Error[1788].CreateEx(TC_Events.Error.Error1788,FALSE,0);
Error[1789].CreateEx(TC_Events.Error.Error1789,FALSE,0);
Error[1790].CreateEx(TC_Events.Error.Error1790,FALSE,0);
Error[1791].CreateEx(TC_Events.Error.Error1791,FALSE,0);
Error[1792].CreateEx(TC_Events.Error.Error1792,FALSE,0);
Error[1793].CreateEx(TC_Events.Error.Error1793,FALSE,0);
Error[1794].CreateEx(TC_Events.Error.Error1794,FALSE,0);
Error[1795].CreateEx(TC_Events.Error.Error1795,FALSE,0);
Error[1796].CreateEx(TC_Events.Error.Error1796,FALSE,0);
Error[1797].CreateEx(TC_Events.Error.Error1797,FALSE,0);
Error[1798].CreateEx(TC_Events.Error.Error1798,FALSE,0);
Error[1799].CreateEx(TC_Events.Error.Error1799,FALSE,0);
Error[1800].CreateEx(TC_Events.Error.Error1800,FALSE,0);
Error[1801].CreateEx(TC_Events.Error.Error1801,FALSE,0);
Error[1802].CreateEx(TC_Events.Error.Error1802,FALSE,0);
Error[1803].CreateEx(TC_Events.Error.Error1803,FALSE,0);
Error[1804].CreateEx(TC_Events.Error.Error1804,FALSE,0);
Error[1805].CreateEx(TC_Events.Error.Error1805,FALSE,0);
Error[1806].CreateEx(TC_Events.Error.Error1806,FALSE,0);
Error[1807].CreateEx(TC_Events.Error.Error1807,FALSE,0);
Error[1808].CreateEx(TC_Events.Error.Error1808,FALSE,0);
Error[1809].CreateEx(TC_Events.Error.Error1809,FALSE,0);
Error[1810].CreateEx(TC_Events.Error.Error1810,FALSE,0);
Error[1811].CreateEx(TC_Events.Error.Error1811,FALSE,0);
Error[1812].CreateEx(TC_Events.Error.Error1812,FALSE,0);
Error[1813].CreateEx(TC_Events.Error.Error1813,FALSE,0);
Error[1814].CreateEx(TC_Events.Error.Error1814,FALSE,0);
Error[1815].CreateEx(TC_Events.Error.Error1815,FALSE,0);
Error[1816].CreateEx(TC_Events.Error.Error1816,FALSE,0);
Error[1817].CreateEx(TC_Events.Error.Error1817,FALSE,0);
Error[1818].CreateEx(TC_Events.Error.Error1818,FALSE,0);
Error[1819].CreateEx(TC_Events.Error.Error1819,FALSE,0);
Error[1820].CreateEx(TC_Events.Error.Error1820,FALSE,0);
Error[1821].CreateEx(TC_Events.Error.Error1821,FALSE,0);
Error[1822].CreateEx(TC_Events.Error.Error1822,FALSE,0);
Error[1823].CreateEx(TC_Events.Error.Error1823,FALSE,0);
Error[1824].CreateEx(TC_Events.Error.Error1824,FALSE,0);
Error[1825].CreateEx(TC_Events.Error.Error1825,FALSE,0);
Error[1826].CreateEx(TC_Events.Error.Error1826,FALSE,0);
Error[1827].CreateEx(TC_Events.Error.Error1827,FALSE,0);
Error[1828].CreateEx(TC_Events.Error.Error1828,FALSE,0);
Error[1829].CreateEx(TC_Events.Error.Error1829,FALSE,0);
Error[1830].CreateEx(TC_Events.Error.Error1830,FALSE,0);
Error[1831].CreateEx(TC_Events.Error.Error1831,FALSE,0);
Error[1832].CreateEx(TC_Events.Error.Error1832,FALSE,0);
Error[1833].CreateEx(TC_Events.Error.Error1833,FALSE,0);
Error[1834].CreateEx(TC_Events.Error.Error1834,FALSE,0);
Error[1835].CreateEx(TC_Events.Error.Error1835,FALSE,0);
Error[1836].CreateEx(TC_Events.Error.Error1836,FALSE,0);
Error[1837].CreateEx(TC_Events.Error.Error1837,FALSE,0);
Error[1838].CreateEx(TC_Events.Error.Error1838,FALSE,0);
Error[1839].CreateEx(TC_Events.Error.Error1839,FALSE,0);
Error[1840].CreateEx(TC_Events.Error.Error1840,FALSE,0);
Error[1841].CreateEx(TC_Events.Error.Error1841,FALSE,0);
Error[1842].CreateEx(TC_Events.Error.Error1842,FALSE,0);
Error[1843].CreateEx(TC_Events.Error.Error1843,FALSE,0);
Error[1844].CreateEx(TC_Events.Error.Error1844,FALSE,0);
Error[1845].CreateEx(TC_Events.Error.Error1845,FALSE,0);
Error[1846].CreateEx(TC_Events.Error.Error1846,FALSE,0);
Error[1847].CreateEx(TC_Events.Error.Error1847,FALSE,0);
Error[1848].CreateEx(TC_Events.Error.Error1848,FALSE,0);
Error[1849].CreateEx(TC_Events.Error.Error1849,FALSE,0);
Error[1850].CreateEx(TC_Events.Error.Error1850,FALSE,0);
Error[1851].CreateEx(TC_Events.Error.Error1851,FALSE,0);
Error[1852].CreateEx(TC_Events.Error.Error1852,FALSE,0);
Error[1853].CreateEx(TC_Events.Error.Error1853,FALSE,0);
Error[1854].CreateEx(TC_Events.Error.Error1854,FALSE,0);
Error[1855].CreateEx(TC_Events.Error.Error1855,FALSE,0);
Error[1856].CreateEx(TC_Events.Error.Error1856,FALSE,0);
Error[1857].CreateEx(TC_Events.Error.Error1857,FALSE,0);
Error[1858].CreateEx(TC_Events.Error.Error1858,FALSE,0);
Error[1859].CreateEx(TC_Events.Error.Error1859,FALSE,0);
Error[1860].CreateEx(TC_Events.Error.Error1860,FALSE,0);
Error[1861].CreateEx(TC_Events.Error.Error1861,FALSE,0);
Error[1862].CreateEx(TC_Events.Error.Error1862,FALSE,0);
Error[1863].CreateEx(TC_Events.Error.Error1863,FALSE,0);
Error[1864].CreateEx(TC_Events.Error.Error1864,FALSE,0);
Error[1865].CreateEx(TC_Events.Error.Error1865,FALSE,0);
Error[1866].CreateEx(TC_Events.Error.Error1866,FALSE,0);
Error[1867].CreateEx(TC_Events.Error.Error1867,FALSE,0);
Error[1868].CreateEx(TC_Events.Error.Error1868,FALSE,0);
Error[1869].CreateEx(TC_Events.Error.Error1869,FALSE,0);
Error[1870].CreateEx(TC_Events.Error.Error1870,FALSE,0);
Error[1871].CreateEx(TC_Events.Error.Error1871,FALSE,0);
Error[1872].CreateEx(TC_Events.Error.Error1872,FALSE,0);
Error[1873].CreateEx(TC_Events.Error.Error1873,FALSE,0);
Error[1874].CreateEx(TC_Events.Error.Error1874,FALSE,0);
Error[1875].CreateEx(TC_Events.Error.Error1875,FALSE,0);
Error[1876].CreateEx(TC_Events.Error.Error1876,FALSE,0);
Error[1877].CreateEx(TC_Events.Error.Error1877,FALSE,0);
Error[1878].CreateEx(TC_Events.Error.Error1878,FALSE,0);
Error[1879].CreateEx(TC_Events.Error.Error1879,FALSE,0);
Error[1880].CreateEx(TC_Events.Error.Error1880,FALSE,0);
Error[1881].CreateEx(TC_Events.Error.Error1881,FALSE,0);
Error[1882].CreateEx(TC_Events.Error.Error1882,FALSE,0);
Error[1883].CreateEx(TC_Events.Error.Error1883,FALSE,0);
Error[1884].CreateEx(TC_Events.Error.Error1884,FALSE,0);
Error[1885].CreateEx(TC_Events.Error.Error1885,FALSE,0);
Error[1886].CreateEx(TC_Events.Error.Error1886,FALSE,0);
Error[1887].CreateEx(TC_Events.Error.Error1887,FALSE,0);
Error[1888].CreateEx(TC_Events.Error.Error1888,FALSE,0);
Error[1889].CreateEx(TC_Events.Error.Error1889,FALSE,0);
Error[1890].CreateEx(TC_Events.Error.Error1890,FALSE,0);
Error[1891].CreateEx(TC_Events.Error.Error1891,FALSE,0);
Error[1892].CreateEx(TC_Events.Error.Error1892,FALSE,0);
Error[1893].CreateEx(TC_Events.Error.Error1893,FALSE,0);
Error[1894].CreateEx(TC_Events.Error.Error1894,FALSE,0);
Error[1895].CreateEx(TC_Events.Error.Error1895,FALSE,0);
Error[1896].CreateEx(TC_Events.Error.Error1896,FALSE,0);
Error[1897].CreateEx(TC_Events.Error.Error1897,FALSE,0);
Error[1898].CreateEx(TC_Events.Error.Error1898,FALSE,0);
Error[1899].CreateEx(TC_Events.Error.Error1899,FALSE,0);
Error[1900].CreateEx(TC_Events.Error.Error1900,FALSE,0);
Error[1901].CreateEx(TC_Events.Error.Error1901,FALSE,0);
Error[1902].CreateEx(TC_Events.Error.Error1902,FALSE,0);
Error[1903].CreateEx(TC_Events.Error.Error1903,FALSE,0);
Error[1904].CreateEx(TC_Events.Error.Error1904,FALSE,0);
Error[1905].CreateEx(TC_Events.Error.Error1905,FALSE,0);
Error[1906].CreateEx(TC_Events.Error.Error1906,FALSE,0);
Error[1907].CreateEx(TC_Events.Error.Error1907,FALSE,0);
Error[1908].CreateEx(TC_Events.Error.Error1908,FALSE,0);
Error[1909].CreateEx(TC_Events.Error.Error1909,FALSE,0);
Error[1910].CreateEx(TC_Events.Error.Error1910,FALSE,0);
Error[1911].CreateEx(TC_Events.Error.Error1911,FALSE,0);
Error[1912].CreateEx(TC_Events.Error.Error1912,FALSE,0);
Error[1913].CreateEx(TC_Events.Error.Error1913,FALSE,0);
Error[1914].CreateEx(TC_Events.Error.Error1914,FALSE,0);
Error[1915].CreateEx(TC_Events.Error.Error1915,FALSE,0);
Error[1916].CreateEx(TC_Events.Error.Error1916,FALSE,0);
Error[1917].CreateEx(TC_Events.Error.Error1917,FALSE,0);
Error[1918].CreateEx(TC_Events.Error.Error1918,FALSE,0);
Error[1919].CreateEx(TC_Events.Error.Error1919,FALSE,0);
Error[1920].CreateEx(TC_Events.Error.Error1920,FALSE,0);
Error[1921].CreateEx(TC_Events.Error.Error1921,FALSE,0);
Error[1922].CreateEx(TC_Events.Error.Error1922,FALSE,0);
Error[1923].CreateEx(TC_Events.Error.Error1923,FALSE,0);
Error[1924].CreateEx(TC_Events.Error.Error1924,FALSE,0);
Error[1925].CreateEx(TC_Events.Error.Error1925,FALSE,0);
Error[1926].CreateEx(TC_Events.Error.Error1926,FALSE,0);
Error[1927].CreateEx(TC_Events.Error.Error1927,FALSE,0);
Error[1928].CreateEx(TC_Events.Error.Error1928,FALSE,0);
Error[1929].CreateEx(TC_Events.Error.Error1929,FALSE,0);
Error[1930].CreateEx(TC_Events.Error.Error1930,FALSE,0);
Error[1931].CreateEx(TC_Events.Error.Error1931,FALSE,0);
Error[1932].CreateEx(TC_Events.Error.Error1932,FALSE,0);
Error[1933].CreateEx(TC_Events.Error.Error1933,FALSE,0);
Error[1934].CreateEx(TC_Events.Error.Error1934,FALSE,0);
Error[1935].CreateEx(TC_Events.Error.Error1935,FALSE,0);
Error[1936].CreateEx(TC_Events.Error.Error1936,FALSE,0);
Error[1937].CreateEx(TC_Events.Error.Error1937,FALSE,0);
Error[1938].CreateEx(TC_Events.Error.Error1938,FALSE,0);
Error[1939].CreateEx(TC_Events.Error.Error1939,FALSE,0);
Error[1940].CreateEx(TC_Events.Error.Error1940,FALSE,0);
Error[1941].CreateEx(TC_Events.Error.Error1941,FALSE,0);
Error[1942].CreateEx(TC_Events.Error.Error1942,FALSE,0);
Error[1943].CreateEx(TC_Events.Error.Error1943,FALSE,0);
Error[1944].CreateEx(TC_Events.Error.Error1944,FALSE,0);
Error[1945].CreateEx(TC_Events.Error.Error1945,FALSE,0);
Error[1946].CreateEx(TC_Events.Error.Error1946,FALSE,0);
Error[1947].CreateEx(TC_Events.Error.Error1947,FALSE,0);
Error[1948].CreateEx(TC_Events.Error.Error1948,FALSE,0);
Error[1949].CreateEx(TC_Events.Error.Error1949,FALSE,0);
Error[1950].CreateEx(TC_Events.Error.Error1950,FALSE,0);
Error[1951].CreateEx(TC_Events.Error.Error1951,FALSE,0);
Error[1952].CreateEx(TC_Events.Error.Error1952,FALSE,0);
Error[1953].CreateEx(TC_Events.Error.Error1953,FALSE,0);
Error[1954].CreateEx(TC_Events.Error.Error1954,FALSE,0);
Error[1955].CreateEx(TC_Events.Error.Error1955,FALSE,0);
Error[1956].CreateEx(TC_Events.Error.Error1956,FALSE,0);
Error[1957].CreateEx(TC_Events.Error.Error1957,FALSE,0);
Error[1958].CreateEx(TC_Events.Error.Error1958,FALSE,0);
Error[1959].CreateEx(TC_Events.Error.Error1959,FALSE,0);
Error[1960].CreateEx(TC_Events.Error.Error1960,FALSE,0);
Error[1961].CreateEx(TC_Events.Error.Error1961,FALSE,0);
Error[1962].CreateEx(TC_Events.Error.Error1962,FALSE,0);
Error[1963].CreateEx(TC_Events.Error.Error1963,FALSE,0);
Error[1964].CreateEx(TC_Events.Error.Error1964,FALSE,0);
Error[1965].CreateEx(TC_Events.Error.Error1965,FALSE,0);
Error[1966].CreateEx(TC_Events.Error.Error1966,FALSE,0);
Error[1967].CreateEx(TC_Events.Error.Error1967,FALSE,0);
Error[1968].CreateEx(TC_Events.Error.Error1968,FALSE,0);
Error[1969].CreateEx(TC_Events.Error.Error1969,FALSE,0);
Error[1970].CreateEx(TC_Events.Error.Error1970,FALSE,0);
Error[1971].CreateEx(TC_Events.Error.Error1971,FALSE,0);
Error[1972].CreateEx(TC_Events.Error.Error1972,FALSE,0);
Error[1973].CreateEx(TC_Events.Error.Error1973,FALSE,0);
Error[1974].CreateEx(TC_Events.Error.Error1974,FALSE,0);
Error[1975].CreateEx(TC_Events.Error.Error1975,FALSE,0);
Error[1976].CreateEx(TC_Events.Error.Error1976,FALSE,0);
Error[1977].CreateEx(TC_Events.Error.Error1977,FALSE,0);
Error[1978].CreateEx(TC_Events.Error.Error1978,FALSE,0);
Error[1979].CreateEx(TC_Events.Error.Error1979,FALSE,0);
Error[1980].CreateEx(TC_Events.Error.Error1980,FALSE,0);
Error[1981].CreateEx(TC_Events.Error.Error1981,FALSE,0);
Error[1982].CreateEx(TC_Events.Error.Error1982,FALSE,0);
Error[1983].CreateEx(TC_Events.Error.Error1983,FALSE,0);
Error[1984].CreateEx(TC_Events.Error.Error1984,FALSE,0);
Error[1985].CreateEx(TC_Events.Error.Error1985,FALSE,0);
Error[1986].CreateEx(TC_Events.Error.Error1986,FALSE,0);
Error[1987].CreateEx(TC_Events.Error.Error1987,FALSE,0);
Error[1988].CreateEx(TC_Events.Error.Error1988,FALSE,0);
Error[1989].CreateEx(TC_Events.Error.Error1989,FALSE,0);
Error[1990].CreateEx(TC_Events.Error.Error1990,FALSE,0);
Error[1991].CreateEx(TC_Events.Error.Error1991,FALSE,0);
Error[1992].CreateEx(TC_Events.Error.Error1992,FALSE,0);
Error[1993].CreateEx(TC_Events.Error.Error1993,FALSE,0);
Error[1994].CreateEx(TC_Events.Error.Error1994,FALSE,0);
Error[1995].CreateEx(TC_Events.Error.Error1995,FALSE,0);
Error[1996].CreateEx(TC_Events.Error.Error1996,FALSE,0);
Error[1997].CreateEx(TC_Events.Error.Error1997,FALSE,0);
Error[1998].CreateEx(TC_Events.Error.Error1998,FALSE,0);
Error[1999].CreateEx(TC_Events.Error.Error1999,FALSE,0);
Error[2000].CreateEx(TC_Events.Error.Error2000,FALSE,0);
END_IF
IF NOT bdone THEN
	bdone:=TRUE;
FOR i:=1 TO 2000 BY 1 DO 
	
IF berror[i] THEN
	berror[i]:=FALSE;
	Error[i].Raise(0);
	temp:=TRUE;
END_IF
END_FOR
bdone:=FALSE;
END_IF

IF reset THEN
	FOR j:=1 TO 2000 BY 1 DO 
	bclear[j]:=FALSE;
	Error[j].Clear(0,TRUE);
	END_FOR
	temp:=false;
END_IF

berror[1]:=Bin1;
berror[2]:=Bin2;
berror[3]:=Bin3;
berror[4]:=Bin4;
berror[101]:=Bin5;
berror[102]:=Bin6;
berror[103]:=Bin7;

(*IF bInit THEN
	bInit:=FALSE;
	Error[1].CreateEx(TC_Events.Error.Error1,TRUE,0);
END_IF

IF bRaise THEN
	bRaise:=FALSE;
	Error[1].Raise(0);
END_IF

IF bclearA THEN
	bclearA := FALSE;
	Error[1].Clear(0,TRUE);
END_IF;*)

END_PROGRAM

(* stored: Version 1.1.0.1, ProductVersion 3.1.4024.11
   POU Error: Id {7f538568-b80b-4a69-ada4-c6183b1c171f}, SpecialFunc None *)
